{attribute 'qualified_only'} // Variable needs to be used with GVL-name

// INT: [-32768, 32767]	
// BOOL: True/False
// %I* assigns next available memory adress in Twincat (In)
VAR_GLOBAL
	// Mode Selection
	bManualMode 		AT %I* : BOOL; // Manual mode controller
	bAutoMode	 		AT %I* : BOOL; // Auto mode controller
	bStartButton		AT %I* : BOOL; // Start button
	bStopButton			AT %I* : BOOL; // Stop button
	
	// Raw Pressure Values
	nRawPa 				AT %I*	: INT; // Pressure cap side
	nRawPb				AT %I*	: INT; // Pressure rod side
	nRawPs				AT %I*	: INT; // Pressure supply
	nRawPaLower			AT %I* 	: INT; // Pressure under counterbalance valve
	
	// Raw Position Values
	nRawPistonPosition 	AT %I*	: INT; // Piston position
	nRawJoystick		AT %I*	: INT; // Joystick Y-position
	nRawFlowSensor		AT %I*	: INT; // Flow sensor
	nRawSpoolPosition	AT %I*	: INT; // Spool position
END_VAR

(* stored: Version 1.1.0.1
   GVL GVL_Inputs: Id {5b9d7628-0828-46aa-93e1-a3aa0cb59901} *)
